FUNCTION_BLOCK ResetGroup  IMPLEMENTS I_Task
VAR
	groupReset			: MC_GroupReset;
	_caGroup			: I_CollisionGroup;
	_Done 				: BOOL;
	_Error				: BOOL;
	_ErrorID			: UDINT;
END_VAR

{analysis -2}

METHOD Abort : BOOL
groupReset.Execute := FALSE;
Abort := TRUE;
END_METHOD

PROPERTY Busy : BOOL
GET
Busy := groupReset.Busy;
END_GET
END_PROPERTY

METHOD Cycle : HRESULT
VAR_INPUT
END_VAR
IF _caGroup = 0 THEN
	cycle := -1;
	RETURN;
END_IF
_Done := groupReset.Done OR _Done;
_Error := groupReset.Error OR _Error;
IF groupReset.ErrorId <> 0 THEN
	_ErrorId := groupReset.ErrorId;
END_IF
groupReset(AxesGroup := _caGroup.GroupRef);
groupReset.Execute := FALSE;
END_METHOD

PROPERTY Done : BOOL
GET
Done := _Done;
END_GET
END_PROPERTY

PROPERTY Error : BOOL
GET
Error := _Error;
END_GET
END_PROPERTY

METHOD Execute : HRESULT
IF groupReset.Execute THEN
	Execute := -1;
	RETURN;
END_IF

IF _caGroup = 0 THEN
	Execute := -2;
	RETURN;
END_IF

groupReset.Execute := TRUE;
END_METHOD

PROPERTY MyCollisionGroup : I_CollisionGroup
GET
MyCollisionGroup := _caGroup;
END_GET
SET
IF MyCollisionGroup <> 0 THEN
	_caGroup := MyCollisionGroup;
END_IF
END_SET
END_PROPERTY

END_FUNCTION_BLOCK

(* stored: Version 1.1.0.1
   POU ResetGroup: Id {c0d0b360-5fec-467e-a65e-491de04b13b3}, SpecialFunc None
   Method Abort: Id {713891a3-4780-46dc-94db-48974077b800}
   Property Busy: Id {082143e7-cb0d-4693-a3c5-aae125aac900}
   Get Get: Id {f3fb4d35-6498-4dc3-9624-a4dbbaa48d6a}
   Method Cycle: Id {60490ba9-dc4f-4168-a59d-a16c9df8b6fb}
   Property Done: Id {c50ed748-a155-44f3-a4e5-da3ebbeffcb4}
   Get Get: Id {896b956f-5079-4ce4-b4a1-b426f3d4396f}
   Property Error: Id {7cc41ac6-6a8c-4645-8a85-d402bdf38d38}
   Get Get: Id {62d28ef8-841d-4940-8890-5b4066e5f424}
   Method Execute: Id {d2d6e3c9-1d94-473e-8bef-e969b6fceb58}
   Property MyCollisionGroup: Id {64ee9bfe-dcea-4ad5-aa89-cde4b64d6f35}
   Get Get: Id {1ff65b10-664c-49ae-bbd9-9f1c1bc2fafc}
   Set Set: Id {7b7d0450-37b2-4626-adf9-a8395e44b7f7} *)
